INTERFACE ITask

METHOD Abort : BOOL
VAR_INPUT
END_VAR
END_METHOD

PROPERTY Busy : bool
GET
END_GET
END_PROPERTY

PROPERTY Done : bool
GET
END_GET
END_PROPERTY

PROPERTY Error : bool
GET
END_GET
END_PROPERTY

END_INTERFACE

(* stored: Version 1.1.0.1, ProductVersion 3.1.4024.11
   Itf ITask: Id {753da03d-a16b-4851-b946-80507957e4ea}
   Method Abort: Id {58dfb800-c837-4fa1-ba5f-77802b4a21e9}
   Property Busy: Id {7b506b51-a48e-4951-a66a-f3a4fad2e014}
   Get Get: Id {893af2fd-0c0a-4421-a795-09e831d3a358}
   Property Done: Id {f41cc815-2884-4cf8-a484-4d14e7adade4}
   Get Get: Id {b34cbf1e-11db-467e-91c9-aa0afac97baf}
   Property Error: Id {2cf05ee7-a555-4b15-9798-5aabce39b467}
   Get Get: Id {6d46dcf2-4281-4caf-b248-8fb4149f403d} *)
